PROGRAM MAIN
VAR
	fbPlantSim   : FB_PlantSimulation;

    fbPressure   : FB_AnalogInput;
    fbBarrelTemp : FB_AnalogInput;
    fbMoldTemp   : FB_AnalogInput;
	fbMachine	 : FB_Machine;
	fbTemperature: FB_TemperatureControl;
	fbInjectionSequence : FB_InjectionSequence;
	fbExtruder	 : FB_Extruder;
	fbMold		 : FB_Mold;
	fbHopper	 : FB_Hopper;
	fbAlarmManager : FB_AlarmManager;
	fbInterlocks : FB_Interlocks;

	// Temporary manual commands for commissioning/testing
	bTestM101_Request   : BOOL := FALSE;
	bTestM102_Request   : BOOL := FALSE;
	bTestM201_l_Request : BOOL := FALSE;
	bTestM201_r_Request : BOOL := FALSE;
	
	 // Vision
    fbVision              : FB_Vision;
    bVisionTestTrigger    : BOOL := FALSE;
    bVisionTestAck        : BOOL := FALSE;
    nVisionTestProductID  : DINT := 1;
    bVisionOffline        : BOOL := FALSE;
	bVisionTimeout : BOOL;
	
	
	nRandomValue : UDINT;
	
	ePreviousSequenceState : E_SequenceState := E_SequenceState.SEQ_IDLE;
	
END_VAR

										// ANALOG INPUT PROCESSING


// Pressure PI101: 0 ... 200 bar
fbPressure(
    nRaw := GVL_IO.PI101_raw,
    fEngMin := 0.0,
    fEngMax := 200.0,
    fValue => GVL_Status.fPressureBar
);


// Barrel temperature TI101: -100 ... 600 °C
fbBarrelTemp(
    nRaw := GVL_IO.TI101_raw,
    fEngMin := -100.0,
    fEngMax := 600.0,
    fValue => GVL_Status.fBarrelTemp
);


// Mold temperature TI201: -100 ... 600 °C
fbMoldTemp(
    nRaw := GVL_IO.TI201_raw,
    fEngMin := -100.0,
    fEngMax := 600.0,
    fValue => GVL_Status.fMoldTemp
);

														// MACHINE MODE CONTROL

fbMachine(
    bStartup := GVL_IO.B_startup,
    bStart := GVL_IO.B_start,
    bStop := GVL_IO.B_stop,
    bShutdown := GVL_IO.B_shutdown,
    bEStop := GVL_IO.B_ES,
    bAck := GVL_IO.B_ack,

    fBarrelTemp := GVL_Status.fBarrelTemp,
    fPressureBar := GVL_Status.fPressureBar,
    bMoldClosed := GVL_IO.ES202,

    bSequenceStopComplete :=
        fbInjectionSequence.bStopComplete,

    eMode => GVL_Status.eMachineMode,
    bMachineReady => GVL_Status.bMachineReady,

    bV2 => GVL_IO.V2,
    bV3 => GVL_IO.V3
);


														// TEMPERATURE CONTROL
fbTemperature(
    bEnable := fbMachine.bTempControlEnable,
	fSetpoint := fbMachine.fTempSetpoint,
    fActualTemp := GVL_Status.fBarrelTemp,

    fHeatingPower => GVL_IO.P_in,
    bCoolingValve => GVL_IO.V1
);

													// AUTOMATIC INJECTION SEQUENCE


fbInjectionSequence(
    bEnable :=
        GVL_Status.eMachineMode =
        E_MachineMode.MODE_RUN,

    bStopRequest := GVL_IO.B_stop,

    bAtFront := GVL_IO.ES101,
    bAtRear := GVL_IO.ES102,

    bMoldOpen := GVL_IO.ES201,
    bMoldClosed := GVL_IO.ES202,

    tCoolingTime := GVL_Config.c_tCoolingTime,

    nProducedParts :=
        GVL_Status.stProduction.nTotalParts,

    nBatchSize :=
        GVL_Config.c_nBatchSize,
		
	bVisionReady :=
    	GVL_Status.stVision.bReady,

	bVisionResultValid :=
    	GVL_Status.stVision.bResultValid,

	bVisionPartOK :=
    	GVL_Status.stVision.bPartOK,
		
	bVisionOffline := fbVision.bOffline,

	bVisionTimeout := fbVision.bTimeout,

    eState => GVL_Status.eSequenceState,
	
	tLastCycleTime =>
        GVL_Status.stProduction.tLastCycleTime
);

	GVL_Status.bCycleActive := fbInjectionSequence.bCycleActive;
	
	GVL_Status.stProduction.fLastCycleTimeSec :=
    	TIME_TO_REAL(GVL_Status.stProduction.tLastCycleTime) / 1000.0;
	

CASE GVL_Status.eMachineMode OF

    E_MachineMode.MODE_INITIAL:
        GVL_Status.sMachineModeText := 'INITIAL';

    E_MachineMode.MODE_STARTUP:
        GVL_Status.sMachineModeText := 'STARTUP';

    E_MachineMode.MODE_STOPPED:
        GVL_Status.sMachineModeText := 'STOPPED';

    E_MachineMode.MODE_RUN:
        GVL_Status.sMachineModeText := 'RUN';

    E_MachineMode.MODE_SHUTDOWN:
        GVL_Status.sMachineModeText := 'SHUTDOWN';

    E_MachineMode.MODE_ESTOP:
        GVL_Status.sMachineModeText := 'E-STOP';

ELSE
    GVL_Status.sMachineModeText := 'UNKNOWN';

END_CASE;





CASE fbInjectionSequence.eState OF

    E_SequenceState.SEQ_IDLE:
        GVL_Status.sSequenceText := 'IDLE';

    E_SequenceState.SEQ_INJECT:
        GVL_Status.sSequenceText := 'INJECT';

    E_SequenceState.SEQ_COOLING:
        GVL_Status.sSequenceText := 'COOLING';

    E_SequenceState.SEQ_DOSING:
        GVL_Status.sSequenceText := 'DOSING';

    E_SequenceState.SEQ_OPEN_MOLD:
        GVL_Status.sSequenceText := 'OPEN MOLD';

    E_SequenceState.SEQ_EJECT:
        GVL_Status.sSequenceText := 'EJECT';

    E_SequenceState.SEQ_CLOSE_MOLD:
        GVL_Status.sSequenceText := 'CLOSE MOLD';

    E_SequenceState.SEQ_VISION_TRIGGER:
        GVL_Status.sSequenceText := 'VISION TRIGGER';

    E_SequenceState.SEQ_VISION_WAIT:
        GVL_Status.sSequenceText := 'VISION WAIT';

    E_SequenceState.SEQ_SORT_PART:
        GVL_Status.sSequenceText := 'SORT PART';

    E_SequenceState.SEQ_COMPLETE:
        GVL_Status.sSequenceText := 'COMPLETE';

ELSE
    GVL_Status.sSequenceText := 'UNKNOWN';

END_CASE;



// =====================================================
// RANDOM VIRTUAL PART GENERATOR
// Select exactly one image when a new cycle enters
// SEQ_INJECT.
// =====================================================

IF GVL_Simulation.bRandomPartMode
   AND
   (fbInjectionSequence.eState = E_SequenceState.SEQ_INJECT)
   AND
   (ePreviousSequenceState <> E_SequenceState.SEQ_INJECT) THEN

    // -------------------------------------------------
    // Generate next pseudo-random number
    // -------------------------------------------------

    GVL_Simulation.nRandomSeed :=
        (GVL_Simulation.nRandomSeed * UDINT#1664525)
        + UDINT#1013904223;

    nRandomValue :=
        GVL_Simulation.nRandomSeed;


    // -------------------------------------------------
    // Map pseudo-random value to dataset index 1..40
    // -------------------------------------------------

    GVL_Simulation.nVisionDatasetIndex :=
        UDINT_TO_INT(
            nRandomValue MOD UDINT#40
        ) + 1;


    // -------------------------------------------------
    // Assign selected image to this molded part
    // -------------------------------------------------

    GVL_Simulation.sVisionImagePath :=
        GVL_Simulation.aVisionDataset[
            GVL_Simulation.nVisionDatasetIndex
        ];

END_IF;


// =====================================================
// STORE CURRENT STATE FOR NEXT PLC SCAN
// This line MUST come after the random-selection logic.
// =====================================================

ePreviousSequenceState :=
    fbInjectionSequence.eState;	
	
	
	
	
											// COUNT PRODUCED PARTS

IF fbInjectionSequence.bPartCompleted THEN

    GVL_Status.stProduction.nTotalParts :=
        GVL_Status.stProduction.nTotalParts + 1;

END_IF;

// Good part counter
IF fbInjectionSequence.bGoodPart THEN

    GVL_Status.stProduction.nGoodParts :=
        GVL_Status.stProduction.nGoodParts + 1;

END_IF;


// Rejected part counter
IF fbInjectionSequence.bRejectedPart THEN

    GVL_Status.stProduction.nRejectedParts :=
        GVL_Status.stProduction.nRejectedParts + 1;

    // Store meaningful reject reason
    IF fbVision.bOffline THEN

        // Vision system unavailable
        GVL_Status.stProduction.nLastDefectCode := UINT#4001;

    ELSIF fbVision.bTimeout THEN

        // Vision inspection timeout
        GVL_Status.stProduction.nLastDefectCode := UINT#4002;

    ELSE

        // Genuine Cognex / simulated inspection defect
        GVL_Status.stProduction.nLastDefectCode :=
            GVL_Status.stVision.nDefectCode;

    END_IF;

END_IF;


// Reject rate
IF GVL_Status.stProduction.nTotalParts > 0 THEN

    GVL_Status.stProduction.fRejectRate :=
        (
            UDINT_TO_REAL(
                GVL_Status.stProduction.nRejectedParts
            )
            /
            UDINT_TO_REAL(
                GVL_Status.stProduction.nTotalParts
            )
        ) * 100.0;

ELSE

    GVL_Status.stProduction.fRejectRate := 0.0;

END_IF;


											// EQUIPMENT CONTROL (Extruder + MOLD)

fbExtruder(
    bRotateCmd :=
        fbMachine.bStartupRotateCmd
        OR fbInjectionSequence.bRotateCmd,

    bInjectCmd :=
        fbInjectionSequence.bInjectCmd,

    bES101 := GVL_IO.ES101,
    bES102 := GVL_IO.ES102
);

fbMold(
    bOpenCmd :=
        fbInjectionSequence.bOpenMoldCmd,

    bCloseCmd :=
        fbMachine.bStartupCloseCmd
        OR fbInjectionSequence.bCloseMoldCmd,

    bES201 := GVL_IO.ES201,
    bES202 := GVL_IO.ES202
);

										// MACHINE INTERLOCKS

fbInterlocks(
    eMode := GVL_Status.eMachineMode,
	bM101_Request := fbExtruder.bRotateRequest,
    bM102_Request := fbExtruder.bInjectRequest,
    bM201_l_Request := fbMold.bOpenRequest,
    bM201_r_Request := fbMold.bCloseRequest,

    bES101 := GVL_IO.ES101,
    bES102 := GVL_IO.ES102,
    bES201 := GVL_IO.ES201,
    bES202 := GVL_IO.ES202,

    bGuardOpen := GVL_IO.S101,

    fPressureBar := GVL_Status.fPressureBar,
    fBarrelTemp := GVL_Status.fBarrelTemp,

    bM101_Enable => GVL_IO.M101,
    bM102_Enable => GVL_IO.M102,
    bM201_l_Enable => GVL_IO.M201_l,
    bM201_r_Enable => GVL_IO.M201_r
);

																	// HOPPER CONTROL

fbHopper(
    eMode := GVL_Status.eMachineMode,

    bLIS101 := GVL_IO.LIS101,
    bLIS102 := GVL_IO.LIS102,

    bAck := GVL_IO.B_ack,

    bFeederRequest => GVL_IO.M301,
    bWarning => GVL_IO.W_hopper
);


// =====================================================
// RANDOM VIRTUAL PART GENERATOR
// Select one image exactly once when entering SEQ_INJECT
// =====================================================

IF GVL_Simulation.bRandomPartMode
   AND
   (fbInjectionSequence.eState = E_SequenceState.SEQ_INJECT)
   AND
   (ePreviousSequenceState <> E_SequenceState.SEQ_INJECT) THEN

    // Generate next pseudo-random number
    GVL_Simulation.nRandomSeed :=
        (GVL_Simulation.nRandomSeed * UDINT#1664525)
        + UDINT#1013904223;

    nRandomValue :=
        GVL_Simulation.nRandomSeed;


    // Convert random value to dataset index 1..40
    GVL_Simulation.nVisionDatasetIndex :=
        UDINT_TO_INT(
            nRandomValue MOD UDINT#40
        ) + 1;


    // Assign selected image to current molded part
    GVL_Simulation.sVisionImagePath :=
        GVL_Simulation.aVisionDataset[
            GVL_Simulation.nVisionDatasetIndex
        ];

END_IF;


// IMPORTANT:
// Store current state only AFTER the random selection check
ePreviousSequenceState :=
    fbInjectionSequence.eState;



																	// VISION SYSTEM
// Temporary simulation / commissioning interface

fbVision(
    bEnable :=
        (GVL_Status.eMachineMode = E_MachineMode.MODE_RUN),

    bTrigger :=
        fbInjectionSequence.bVisionTrigger,

    bAck :=
        fbInjectionSequence.bVisionAck,

    bFaultAck :=
        GVL_IO.B_ack,

    bForceOffline :=
        GVL_Simulation.bForceVisionOffline,

    bForceTimeout :=
        GVL_Simulation.bForceVisionTimeout,

    nProductID :=
        UDINT_TO_DINT(
            GVL_Status.stProduction.nTotalParts + 1
        ),
		
	sImagePath :=
		GVL_Simulation.sVisionImagePath,

    stResult =>
        GVL_Status.stVision,

    bOffline =>
        bVisionOffline,
		
	bTimeout =>
        bVisionTimeout
);

																	// ALARM MANAGEMENT


fbAlarmManager(
    eMode := GVL_Status.eMachineMode,

    bHopperLowTimeout :=
        fbHopper.bLowLevelTimeout,

    bHopperFillTimeout :=
        fbHopper.bFillTimeout,

    fBarrelTemp :=
        GVL_Status.fBarrelTemp,

    fPressureBar :=
        GVL_Status.fPressureBar,

    bGuardOpen :=
        GVL_IO.S101,

    bEStop :=
        GVL_IO.B_ES,

    bVisionOffline :=
        bVisionOffline,

    bVisionTimeout :=
		fbVision.bTimeout,

    bAck :=
        GVL_IO.B_ack,

    bFaultActive =>
        GVL_Status.bFaultActive,

    eActiveAlarm =>
        GVL_Status.eActiveAlarm
);

CASE GVL_Status.eActiveAlarm OF

    E_AlarmID.ALARM_NONE:
        GVL_Status.sActiveAlarmText := 'NONE';

    E_AlarmID.ALARM_VISION_OFFLINE:
        GVL_Status.sActiveAlarmText := 'VISION OFFLINE';

    E_AlarmID.ALARM_VISION_TIMEOUT:
        GVL_Status.sActiveAlarmText := 'VISION TIMEOUT';

ELSE
    GVL_Status.sActiveAlarmText := 'ALARM ACTIVE';

END_CASE;

											// PLANT SIMULATION

fbPlantSim(
    bEnable := GVL_Simulation.bSimulationEnabled,

    bM101 := GVL_IO.M101,
    bM102 := GVL_IO.M102,
    bM201_l := GVL_IO.M201_l,
    bM201_r := GVL_IO.M201_r,
    bM301 := GVL_IO.M301,

    bV1 := GVL_IO.V1,
    bV2 := GVL_IO.V2,
    bV3 := GVL_IO.V3,

    fHeaterPower := GVL_IO.P_in,

    eMode := GVL_Status.eMachineMode,

    bES101 => GVL_IO.ES101,
    bES102 => GVL_IO.ES102,
    bES201 => GVL_IO.ES201,
    bES202 => GVL_IO.ES202,

    bLIS101 => GVL_IO.LIS101,
    bLIS102 => GVL_IO.LIS102,

    nPI101Raw => GVL_IO.PI101_raw,
    nTI101Raw => GVL_IO.TI101_raw,
    nTI201Raw => GVL_IO.TI201_raw
);

//PRG_VisionTest();

END_PROGRAM

(* stored: Version 1.1.0.1, ProductVersion 3.1.4024.16
   POU MAIN: Id {8ea770d7-29d7-4617-838f-87fb45ad0588}, SpecialFunc None *)
